PROGRAM prgPumpControl
VAR
	bStart_PB	:BOOL;
	bStop_PB	:BOOL;
	bPumpRelay	:BOOL;
END_VAR

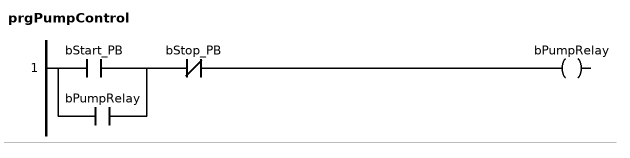
// NETWORK 1
bPumpRelay := (bStart_PB OR bPumpRelay) AND NOT bStop_PB;

END_PROGRAM

(* stored: Version 1.1.0.1, ProductVersion 3.1.4024.13
   POU prgPumpControl: Id {d2f58661-8347-452d-a97f-8736c8fe0145}, SpecialFunc None *)
